# EPICS autosave request: iocBoot/iocThorLabsDFM/auto_settings.req
file "ThorLabsDFM_settings.req", P=$(P), R=$(R)
